FUNCTION_BLOCK FB_test
VAR_INPUT
END_VAR
VAR_OUTPUT
END_VAR
VAR
END_VAR

END_FUNCTION_BLOCK

(* stored: Version 1.1.0.1, ProductVersion 3.1.4024.11
   POU FB_test: Id {3d4c6f9d-e028-4b31-a721-174ac5903662}, SpecialFunc None *)
